KUKA KRL program: Return_Home.src, Return_Home.dat

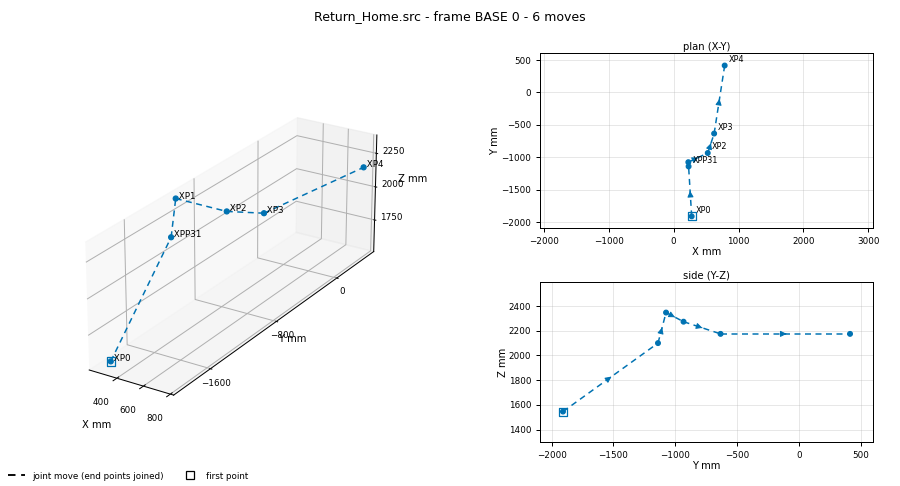
[picture p0: tool path of Return_Home.src in frame BASE 0, 6 of 6 moves have a stored position in this frame; points joined in program order, loops and branches not executed]
--- Return_Home.src ---
&ACCESS RVP13
&REL 42
&COMMENT Return to Home V3.0 Date:12/10/2010
DEF RETURN_HOME (AREA_NR :IN,RETHME_IN :IN)
;================================================
; MODELO   : C-520
; IE GRUPO : 5J
; ESTACION : 85
; ROBOT    : 85r01
; FUNCTION : Return To Home Position
;================================================
;FOLD INI
  INT AREA_NR
  INT RETHME_IN

  IF RETHME_IN==0 THEN
    REPEAT
      EMPTY_MSG={MSG_T: VALID FALSE,RELEASE FALSE,TYP #NOTIFY,MODUL[] " ",KEY[] " ",PARAM_TYP #VALUE,PARAM[] " ",DLG_FORMAT[] " ",ANSWER 0}
      $MSG_T={MSG_T: VALID FALSE,RELEASE FALSE,TYP #QUIT,MODUL[] "Return To Home",KEY[] "Return to waitpos path not configured !!!",PARAM_TYP #KEY,PARAM[] " ",DLG_FORMAT[] " ",ANSWER 0}
      WAIT SEC 1.0
      $MSG_T.VALID=TRUE
      HALT
    UNTIL (RETHME_IN<2) AND (RETHME_IN>0)
  ENDIF

  IF (AREA_NR>8) OR (AREA_NR<1) THEN
    REPEAT
      EMPTY_MSG={MSG_T: VALID FALSE,RELEASE FALSE,TYP #NOTIFY,MODUL[] " ",KEY[] " ",PARAM_TYP #VALUE,PARAM[] " ",DLG_FORMAT[] " ",ANSWER 0}
      $MSG_T={MSG_T: VALID FALSE,RELEASE FALSE,TYP #QUIT,MODUL[] "Return To Home",KEY[] "Area Number Not Valid",PARAM_TYP #KEY,PARAM[] " ",DLG_FORMAT[] " ",ANSWER 0}
      WAIT SEC 1.0
      $MSG_T.VALID=TRUE
      HALT
    UNTIL (AREA_NR<9) AND (AREA_NR>0)
  ENDIF
  ;ENDFOLD

;================================================

SWITCH AREA_NR

CASE 1  ;AREA 1

;Teach here positions from wait area to Waitpos
;check robot movement for collision with other robots

;FOLD PTP P0 CONT Vel=15 % PDAT0 Tool[0] Base[0];%{PE}%R 5.6.13,%MKUKATPBASIS,%CMOVE,%VPTP,%P 1:PTP, 2:P0, 3:C_PTP, 5:15, 7:PDAT0
$BWDSTART=FALSE
PDAT_ACT=PPDAT0
FDAT_ACT=FP0
BAS(#PTP_PARAMS,15)
PTP XP0 C_PTP
;ENDFOLD
;FOLD PTP PP31 Vel=15 % PDAT1 Tool[1]:weld Base[0];%{PE}%R 5.6.13,%MKUKATPBASIS,%CMOVE,%VPTP,%P 1:PTP, 2:PP31, 3:, 5:15, 7:PDAT1
$BWDSTART=FALSE
PDAT_ACT=PPDAT1
FDAT_ACT=FPP31
BAS(#PTP_PARAMS,15)
PTP XPP31
;ENDFOLD
;FOLD PTP P1 Vel=100 % PDAT2 Tool[1]:weld Base[0];%{PE}%R 5.6.13,%MKUKATPBASIS,%CMOVE,%VPTP,%P 1:PTP, 2:P1, 3:, 5:100, 7:PDAT2
$BWDSTART=FALSE
PDAT_ACT=PPDAT2
FDAT_ACT=FP1
BAS(#PTP_PARAMS,100)
PTP XP1
;ENDFOLD
;FOLD PTP P2 Vel=100 % PDAT3 Tool[1]:weld Base[0];%{PE}%R 5.6.13,%MKUKATPBASIS,%CMOVE,%VPTP,%P 1:PTP, 2:P2, 3:, 5:100, 7:PDAT3
$BWDSTART=FALSE
PDAT_ACT=PPDAT3
FDAT_ACT=FP2
BAS(#PTP_PARAMS,100)
PTP XP2
;ENDFOLD
;FOLD PTP P3 Vel=100 % PDAT4 Tool[1]:weld Base[0];%{PE}%R 5.6.13,%MKUKATPBASIS,%CMOVE,%VPTP,%P 1:PTP, 2:P3, 3:, 5:100, 7:PDAT4
$BWDSTART=FALSE
PDAT_ACT=PPDAT4
FDAT_ACT=FP3
BAS(#PTP_PARAMS,100)
PTP XP3
;ENDFOLD
;FOLD PTP P4 Vel=100 % PDAT5 Tool[1]:weld Base[0];%{PE}%R 5.6.13,%MKUKATPBASIS,%CMOVE,%VPTP,%P 1:PTP, 2:P4, 3:, 5:100, 7:PDAT5
$BWDSTART=FALSE
PDAT_ACT=PPDAT5
FDAT_ACT=FP4
BAS(#PTP_PARAMS,100)
PTP XP4
;ENDFOLD
;Delete if movement is used

CASE 2  ;AREA 2

;Teach here positions from wait area to Waitpos
;check robot movement for collision with other robots

;Delete if movement is used
WAIT FOR FALSE

CASE 3  ;AREA 3

;Teach here positions from wait area to Waitpos
;check robot movement for collision with other robots

;Delete if movement is used
WAIT FOR FALSE

CASE 4  ;AREA 4

;Teach here positions from wait area to Waitpos
;check robot movement for collision with other robots

;Delete if movement is used
WAIT FOR FALSE

CASE 5  ;AREA 5

;Teach here positions from wait area to Waitpos
;check robot movement for collision with other robots

;Delete if movement is used
WAIT FOR FALSE

CASE 6  ;AREA 6

;Teach here positions from wait area to Waitpos
;check robot movement for collision with other robots

;Delete if movement is used
WAIT FOR FALSE

CASE 7  ;AREA 7

;Teach here positions from wait area to Waitpos
;check robot movement for collision with other robots

;Delete if movement is used
WAIT FOR FALSE

CASE 8  ;AREA 8

;Teach here positions from wait area to Waitpos
;check robot movement for collision with other robots

;Delete if movement is used
WAIT FOR FALSE

DEFAULT
    REPEAT
      EMPTY_MSG={MSG_T: VALID FALSE,RELEASE FALSE,TYP #NOTIFY,MODUL[] " ",KEY[] " ",PARAM_TYP #VALUE,PARAM[] " ",DLG_FORMAT[] " ",ANSWER 0}
      $MSG_T={MSG_T: VALID FALSE,RELEASE FALSE,TYP #QUIT,MODUL[] "Return To Waitpos",KEY[] "Area Number Not Valid",PARAM_TYP #KEY,PARAM[] " ",DLG_FORMAT[] " ",ANSWER 0}
      WAIT SEC 1.0
      $MSG_T.VALID=TRUE
      HALT
    UNTIL (AREA_NR<9) AND (AREA_NR>0)
ENDSWITCH
END

--- Return_Home.dat ---
&ACCESS RVP13
&REL 42
&COMMENT Return to Home V3.0 Date:12/10/2010
DEFDAT  RETURN_HOME
;FOLD EXTERNAL DECLARATIONS;%{PE}%V3.2.0,%MKUKATPBASIS,%CEXT,%VCOMMON,%P
;FOLD BAS EXT;%{PE}%V3.2.0,%MKUKATPBASIS,%CEXT,%VEXT,%P
EXT  BAS (BAS_COMMAND  :IN,REAL  :IN )
DECL INT SUCCESS
;ENDFOLD
;FOLD GRIPPER EXT;%{E}%V3.2.0,%MKUKATPGRIPPER,%CEXT,%VEXT,%P
EXT  H50 (INT  :IN,INT  :IN,INT  :IN,GRP_TYP  :IN )
;ENDFOLD
;FOLD SPOT EXT;%{E}%V3.2.0,%MKUKATPSPOT,%CEXT,%VEXT,%P
EXT  USERSPOT (S_COMMAND  :IN,SPOT_TYPE  :IN )
;ENDFOLD
;FOLD USER EXT;%{E}%V3.2.0,%MKUKATPUSER,%CEXT,%VEXT,%P
;Make here your modifications
;ENDFOLD
;ENDFOLD

DECL BASIS_SUGG_T LAST_BASIS={POINT1[] "P4                      ",POINT2[] "P4                      ",CP_PARAMS[] "CPDAT0                  ",PTP_PARAMS[] "PDAT5                   ",CONT[] "                        ",CP_VEL[] "2.0                     ",PTP_VEL[] "100                     ",SYNC_PARAMS[] "SYNCDAT                 ",SPL_NAME[] "S0                      "}
DECL PDAT PPDAT0={VEL 100.0,ACC 100.0,APO_DIST 100.0,APO_MODE #CPTP}
DECL E6POS XP0={X 278.475586,Y -1908.98804,Z 1545.66394,A -179.522293,B 44.2849312,C -178.149902,S 2,T 10,E1 0.0,E2 0.0,E3 0.0,E4 0.0,E5 0.0,E6 0.0}
DECL FDAT FP0={TOOL_NO 0,BASE_NO 0,IPO_FRAME #BASE,POINT2[] " ",TQ_STATE FALSE}
DECL PDAT PPDAT1={VEL 100.0,ACC 100.0,APO_DIST 100.0}
DECL E6POS XPP31={X 230.806702,Y -1139.68506,Z 2100.01196,A -88.1130219,B 61.2092094,C -87.0944672,S 2,T 10,E1 0.0,E2 0.0,E3 0.0,E4 0.0,E5 0.0,E6 0.0}
DECL FDAT FPP31={TOOL_NO 1,BASE_NO 0,IPO_FRAME #BASE,POINT2[] " ",TQ_STATE FALSE}
DECL PDAT PPDAT2={VEL 100.0,ACC 100.0,APO_DIST 100.0}
DECL E6POS XP1={X 226.764099,Y -1074.44299,Z 2347.30688,A -87.7077637,B 50.4100189,C -86.6066971,S 2,T 10,E1 0.0,E2 0.0,E3 0.0,E4 0.0,E5 0.0,E6 0.0}
DECL FDAT FP1={TOOL_NO 1,BASE_NO 0,IPO_FRAME #BASE,POINT2[] " ",TQ_STATE FALSE}
DECL PDAT PPDAT3={VEL 100.0,ACC 100.0,APO_DIST 100.0}
DECL E6POS XP2={X 526.068909,Y -932.987793,Z 2273.41699,A -69.0727921,B 61.6084595,C -94.4467697,S 2,T 10,E1 0.0,E2 0.0,E3 0.0,E4 0.0,E5 0.0,E6 0.0}
DECL FDAT FP2={TOOL_NO 1,BASE_NO 0,IPO_FRAME #BASE,POINT2[] " ",TQ_STATE FALSE}
DECL PDAT PPDAT4={VEL 100.0,ACC 100.0,APO_DIST 100.0}
DECL E6POS XP3={X 624.439392,Y -633.425476,Z 2174.77002,A -55.7007103,B 61.2513084,C -94.4497833,S 2,T 10,E1 0.0,E2 0.0,E3 0.0,E4 0.0,E5 0.0,E6 0.0}
DECL FDAT FP3={TOOL_NO 1,BASE_NO 0,IPO_FRAME #BASE,POINT2[] " ",TQ_STATE FALSE}
DECL PDAT PPDAT5={VEL 100.0,ACC 100.0,APO_DIST 100.0}
DECL E6POS XP4={X 786.753174,Y 414.935913,Z 2174.77002,A 17.5158997,B 61.2513084,C -94.4497833,S 2,T 11,E1 0.0,E2 0.0,E3 0.0,E4 0.0,E5 0.0,E6 0.0}
DECL FDAT FP4={TOOL_NO 1,BASE_NO 0,IPO_FRAME #BASE,POINT2[] " ",TQ_STATE FALSE}
ENDDAT
